Omron CX-Programmer project NewProject (CX-Programmer 9.03)

# PLC NewPLC1: CP1L L

## Global symbols (name address type ; comment)
1.02 BOOL  ; MV1
1.01 BOOL  ; MV2
1.00 BOOL  ; M
0.00 BOOL  ; START
0.01 BOOL  ; STOP
0.10 BOOL  ; TLB2
0.11 BOOL  ; TLB1

## Program NewProgram1 (cyclic task 0)

### Section Section1

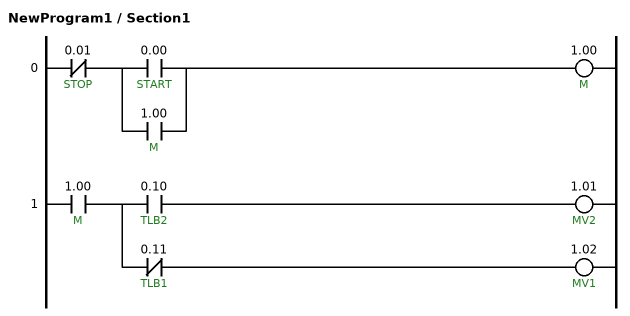
; rung 0
LDNOT 0.01  ; STOP
LD 0.00  ; START
OR 1.00  ; M
ANDLD
OUT 1.00  ; M
; rung 1
LD 1.00  ; M
OUT TR0
AND 0.10  ; TLB2
OUT 1.01  ; MV2
LD TR0
ANDNOT 0.11  ; TLB1
OUT 1.02  ; MV1

### Section END
; rung 0
END(001)